ORGANIZATION_BLOCK 主程序:OB1
TITLE=程序注释
BEGIN
Network 1 // 网络标题
// 网络注释
LD     I0.0
MOVB   16#0, VB100
MOVB   16#05, VB101
MOVB   16#30, VB102
MOVB   16#21, VB103
MOVB   16#0, VB104
MOVB   16#0, VB105
MOVB   16#0, VB106
MOVB   16#03, VB107
TODW   VB100
END_ORGANIZATION_BLOCK
SUBROUTINE_BLOCK SBR_0:SBR0
TITLE=子程序注释
BEGIN
Network 1 // 网络标题
// 网络注释
END_SUBROUTINE_BLOCK
INTERRUPT_BLOCK INT_0:INT0
TITLE=中断程序注释
BEGIN
Network 1 // 网络标题
// 网络注释
END_INTERRUPT_BLOCK
